// TIA Portal V20 export
TYPE "EsopZone"
// stored: Access Published, Namespace Global
   STRUCT
      "1" : Bool;
      "2" : Bool;
   END_STRUCT;
END_TYPE
